// Mitsubishi GX Works2 project: 230930-001- exercicios-0-2   PLC: Q03UDV

// task Task_01 (event TRUE, interval 0, priority 31): POU_01

PROGRAM POU_01
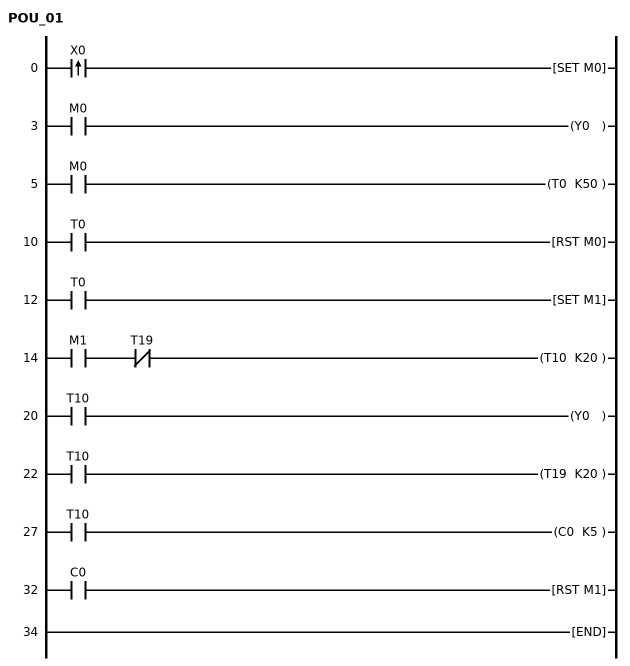
0     LDP     X0
      SET     M0
3     LD      M0
      OUT     Y0
5     LD      M0
      OUT     T0 K50
10    LD      T0
      RST     M0
12    LD      T0
      SET     M1
14    LD      M1
      ANI     T19
      OUT     T10 K20
20    LD      T10
      OUT     Y0
22    LD      T10
      OUT     T19 K20
27    LD      T10
      OUT     C0 K5
32    LD      C0
      RST     M1
34    END
END_PROGRAM
